{attribute 'qualified_only'}
{attribute 'strict'}
TYPE E_StopState :
(
	Init, 
	StopMotor, 
	CloseSolenoids, 
	Delay, 
	ResetMotor, 
	MoveHome, 
	Done
);
END_TYPE

(* stored: Version 1.1.0.1, ProductVersion 3.1.4024.15
   DUT E_StopState: Id {fcbec684-89b8-4cf9-aaeb-669e1941694b} *)
